METHOD Init_RattlingKM
VAR_INPUT
END_VAR
VAR

END_VAR
                          in_0303_05_1_ixSection1_OverheatAlarm(
	ixSignal:= _0303_05_1_ixSection1_OverheatAlarm, 
	itInputTime:= tRattlingDelay, 
	itRattling_count_reset:= , 
	ixResetAlarm:= , 
	qxSignal=> , 
	qxRattlingAlarm=> );
in_0303_05_1_ixSection1_OverheatWarning(
	ixSignal:= _0303_05_1_ixSection1_OverheatWarning, 
	itInputTime:= tRattlingDelay, 
	itRattling_count_reset:= , 
	ixResetAlarm:= , 
	qxSignal=> , 
	qxRattlingAlarm=> );
in_0303_05_1_ixVFD_Failure(
	ixSignal:= _0303_05_1_ixVFD_Failure, 
	itInputTime:= tRattlingDelay, 
	itRattling_count_reset:= , 
	ixResetAlarm:= , 
	qxSignal=> , 
	qxRattlingAlarm=> );
in_0303_05_1_ixVFD_InWork(
	ixSignal:= _0303_05_1_ixVFD_InWork, 
	itInputTime:= tRattlingDelay, 
	itRattling_count_reset:= , 
	ixResetAlarm:= , 
	qxSignal=> , 
	qxRattlingAlarm=> );
in_0303_05_1_ixVFD_Manual(
	ixSignal:= _0303_05_1_ixVFD_Manual, 
	itInputTime:= tRattlingDelay, 
	itRattling_count_reset:= , 
	ixResetAlarm:= , 
	qxSignal=> , 
	qxRattlingAlarm=> );
in_0303_05_1_ixVFD_Ready(
	ixSignal:= _0303_05_1_ixVFD_Ready, 
	itInputTime:= tRattlingDelay, 
	itRattling_count_reset:= , 
	ixResetAlarm:= , 
	qxSignal=> , 
	qxRattlingAlarm=> );
in_0303_05_2_ixSection1_OverheatAlarm(
	ixSignal:= _0303_05_2_ixSection1_OverheatAlarm, 
	itInputTime:= tRattlingDelay, 
	itRattling_count_reset:= , 
	ixResetAlarm:= , 
	qxSignal=> , 
	qxRattlingAlarm=> );
in_0303_05_2_ixSection1_OverheatWarning(
	ixSignal:= _0303_05_2_ixSection1_OverheatWarning, 
	itInputTime:= tRattlingDelay, 
	itRattling_count_reset:= , 
	ixResetAlarm:= , 
	qxSignal=> , 
	qxRattlingAlarm=> );
in_0303_05_2_ixVFD_Failure(
	ixSignal:= _0303_05_2_ixVFD_Failure, 
	itInputTime:= tRattlingDelay, 
	itRattling_count_reset:= , 
	ixResetAlarm:= , 
	qxSignal=> , 
	qxRattlingAlarm=> );
in_0303_05_2_ixVFD_InWork(
	ixSignal:= _0303_05_2_ixVFD_InWork, 
	itInputTime:= tRattlingDelay, 
	itRattling_count_reset:= , 
	ixResetAlarm:= , 
	qxSignal=> , 
	qxRattlingAlarm=> );
in_0303_05_2_ixVFD_Manual(
	ixSignal:= _0303_05_2_ixVFD_Manual, 
	itInputTime:= tRattlingDelay, 
	itRattling_count_reset:= , 
	ixResetAlarm:= , 
	qxSignal=> , 
	qxRattlingAlarm=> );
in_0303_05_2_ixVFD_Ready(
	ixSignal:= _0303_05_2_ixVFD_Ready, 
	itInputTime:= tRattlingDelay, 
	itRattling_count_reset:= , 
	ixResetAlarm:= , 
	qxSignal=> , 
	qxRattlingAlarm=> );
in_0303_05_1KM8_ixStatusOn(
	ixSignal:= _0303_05_1KM8_ixStatusOn, 
	itInputTime:= tRattlingDelay, 
	itRattling_count_reset:= , 
	ixResetAlarm:= , 
	qxSignal=> , 
	qxRattlingAlarm=> );
in_0303_05_2KM8_ixStatusOn(
	ixSignal:= _0303_05_2KM8_ixStatusOn, 
	itInputTime:= tRattlingDelay, 
	itRattling_count_reset:= , 
	ixResetAlarm:= , 
	qxSignal=> , 
	qxRattlingAlarm=> );
in_0303_05_BY01_ixKM_PosClosed(
	ixSignal:= _0303_05_BY01_ixKM_PosClosed, 
	itInputTime:= tRattlingDelay, 
	itRattling_count_reset:= , 
	ixResetAlarm:= , 
	qxSignal=> , 
	qxRattlingAlarm=> );
in_0303_05_BY01_ixKM_PosOpen(
	ixSignal:= _0303_05_BY01_ixKM_PosOpen, 
	itInputTime:= tRattlingDelay, 
	itRattling_count_reset:= , 
	ixResetAlarm:= , 
	qxSignal=> , 
	qxRattlingAlarm=> );
in_0303_05_BY01_ixShutter_PosClosed(
	ixSignal:= _0303_05_BY01_ixShutter_PosClosed, 
	itInputTime:= tRattlingDelay, 
	itRattling_count_reset:= , 
	ixResetAlarm:= , 
	qxSignal=> , 
	qxRattlingAlarm=> );
in_0303_05_BY01_ixShutter_PosOpen(
	ixSignal:= _0303_05_BY01_ixShutter_PosOpen, 
	itInputTime:= tRattlingDelay, 
	itRattling_count_reset:= , 
	ixResetAlarm:= , 
	qxSignal=> , 
	qxRattlingAlarm=> );
in_0303_05_BY01_ixShutter_StatusError(
	ixSignal:= _0303_05_BY01_ixShutter_StatusError, 
	itInputTime:= tRattlingDelay, 
	itRattling_count_reset:= , 
	ixResetAlarm:= , 
	qxSignal=> , 
	qxRattlingAlarm=> );
in_0303_05_BY01_ixShutter_StatusReady(
	ixSignal:= _0303_05_BY01_ixShutter_StatusReady, 
	itInputTime:= tRattlingDelay, 
	itRattling_count_reset:= , 
	ixResetAlarm:= , 
	qxSignal=> , 
	qxRattlingAlarm=> );
in_0303_05_BY02_ixKM_PosClosed(
	ixSignal:= _0303_05_BY02_ixKM_PosClosed, 
	itInputTime:= tRattlingDelay, 
	itRattling_count_reset:= , 
	ixResetAlarm:= , 
	qxSignal=> , 
	qxRattlingAlarm=> );
in_0303_05_BY02_ixKM_PosOpen(
	ixSignal:= _0303_05_BY02_ixKM_PosOpen, 
	itInputTime:= tRattlingDelay, 
	itRattling_count_reset:= , 
	ixResetAlarm:= , 
	qxSignal=> , 
	qxRattlingAlarm=> );
in_0303_05_BY02_ixShutter_PosClosed(
	ixSignal:= _0303_05_BY02_ixShutter_PosClosed, 
	itInputTime:= tRattlingDelay, 
	itRattling_count_reset:= , 
	ixResetAlarm:= , 
	qxSignal=> , 
	qxRattlingAlarm=> );
in_0303_05_BY02_ixShutter_PosOpen(
	ixSignal:= _0303_05_BY02_ixShutter_PosOpen, 
	itInputTime:= tRattlingDelay, 
	itRattling_count_reset:= , 
	ixResetAlarm:= , 
	qxSignal=> , 
	qxRattlingAlarm=> );
in_0303_05_BY02_ixShutter_StatusError(
	ixSignal:= _0303_05_BY02_ixShutter_StatusError, 
	itInputTime:= tRattlingDelay, 
	itRattling_count_reset:= , 
	ixResetAlarm:= , 
	qxSignal=> , 
	qxRattlingAlarm=> );
in_0303_05_BY02_ixShutter_StatusReady(
	ixSignal:= _0303_05_BY02_ixShutter_StatusReady, 
	itInputTime:= tRattlingDelay, 
	itRattling_count_reset:= , 
	ixResetAlarm:= , 
	qxSignal=> , 
	qxRattlingAlarm=> );
in_0303_05_BY03_ixKM_PosClosed(
	ixSignal:= _0303_05_BY03_ixKM_PosClosed, 
	itInputTime:= tRattlingDelay, 
	itRattling_count_reset:= , 
	ixResetAlarm:= , 
	qxSignal=> , 
	qxRattlingAlarm=> );
in_0303_05_BY03_ixKM_PosOpen(
	ixSignal:= _0303_05_BY03_ixKM_PosOpen, 
	itInputTime:= tRattlingDelay, 
	itRattling_count_reset:= , 
	ixResetAlarm:= , 
	qxSignal=> , 
	qxRattlingAlarm=> );
in_0303_05_BY03_ixShutter_PosClosed(
	ixSignal:= _0303_05_BY03_ixShutter_PosClosed, 
	itInputTime:= tRattlingDelay, 
	itRattling_count_reset:= , 
	ixResetAlarm:= , 
	qxSignal=> , 
	qxRattlingAlarm=> );
in_0303_05_BY03_ixShutter_PosOpen(
	ixSignal:= _0303_05_BY03_ixShutter_PosOpen, 
	itInputTime:= tRattlingDelay, 
	itRattling_count_reset:= , 
	ixResetAlarm:= , 
	qxSignal=> , 
	qxRattlingAlarm=> );
in_0303_05_BY03_ixShutter_StatusError(
	ixSignal:= _0303_05_BY03_ixShutter_StatusError, 
	itInputTime:= tRattlingDelay, 
	itRattling_count_reset:= , 
	ixResetAlarm:= , 
	qxSignal=> , 
	qxRattlingAlarm=> );
in_0303_05_BY03_ixShutter_StatusReady(
	ixSignal:= _0303_05_BY03_ixShutter_StatusReady, 
	itInputTime:= tRattlingDelay, 
	itRattling_count_reset:= , 
	ixResetAlarm:= , 
	qxSignal=> , 
	qxRattlingAlarm=> );
in_0303_05_BY04_ixKM_PosClosed(
	ixSignal:= _0303_05_BY04_ixKM_PosClosed, 
	itInputTime:= tRattlingDelay, 
	itRattling_count_reset:= , 
	ixResetAlarm:= , 
	qxSignal=> , 
	qxRattlingAlarm=> );
in_0303_05_BY04_ixKM_PosOpen(
	ixSignal:= _0303_05_BY04_ixKM_PosOpen, 
	itInputTime:= tRattlingDelay, 
	itRattling_count_reset:= , 
	ixResetAlarm:= , 
	qxSignal=> , 
	qxRattlingAlarm=> );
in_0303_05_BY04_ixShutter_PosClosed(
	ixSignal:= _0303_05_BY04_ixShutter_PosClosed, 
	itInputTime:= tRattlingDelay, 
	itRattling_count_reset:= , 
	ixResetAlarm:= , 
	qxSignal=> , 
	qxRattlingAlarm=> );
in_0303_05_BY04_ixShutter_PosOpen(
	ixSignal:= _0303_05_BY04_ixShutter_PosOpen, 
	itInputTime:= tRattlingDelay, 
	itRattling_count_reset:= , 
	ixResetAlarm:= , 
	qxSignal=> , 
	qxRattlingAlarm=> );
in_0303_05_BY04_ixShutter_StatusError(
	ixSignal:= _0303_05_BY04_ixShutter_StatusError, 
	itInputTime:= tRattlingDelay, 
	itRattling_count_reset:= , 
	ixResetAlarm:= , 
	qxSignal=> , 
	qxRattlingAlarm=> );
in_0303_05_BY04_ixShutter_StatusReady(
	ixSignal:= _0303_05_BY04_ixShutter_StatusReady, 
	itInputTime:= tRattlingDelay, 
	itRattling_count_reset:= , 
	ixResetAlarm:= , 
	qxSignal=> , 
	qxRattlingAlarm=> );
in_0303_05_BY05_ixKM_PosClosed(
	ixSignal:= _0303_05_BY05_ixKM_PosClosed, 
	itInputTime:= tRattlingDelay, 
	itRattling_count_reset:= , 
	ixResetAlarm:= , 
	qxSignal=> , 
	qxRattlingAlarm=> );
in_0303_05_BY05_ixKM_PosOpen(
	ixSignal:= _0303_05_BY05_ixKM_PosOpen, 
	itInputTime:= tRattlingDelay, 
	itRattling_count_reset:= , 
	ixResetAlarm:= , 
	qxSignal=> , 
	qxRattlingAlarm=> );
in_0303_05_BY05_ixShutter_PosClosed(
	ixSignal:= _0303_05_BY05_ixShutter_PosClosed, 
	itInputTime:= tRattlingDelay, 
	itRattling_count_reset:= , 
	ixResetAlarm:= , 
	qxSignal=> , 
	qxRattlingAlarm=> );
in_0303_05_BY05_ixShutter_PosOpen(
	ixSignal:= _0303_05_BY05_ixShutter_PosOpen, 
	itInputTime:= tRattlingDelay, 
	itRattling_count_reset:= , 
	ixResetAlarm:= , 
	qxSignal=> , 
	qxRattlingAlarm=> );
in_0303_05_BY05_ixShutter_StatusError(
	ixSignal:= _0303_05_BY05_ixShutter_StatusError, 
	itInputTime:= tRattlingDelay, 
	itRattling_count_reset:= , 
	ixResetAlarm:= , 
	qxSignal=> , 
	qxRattlingAlarm=> );
in_0303_05_BY05_ixShutter_StatusReady(
	ixSignal:= _0303_05_BY05_ixShutter_StatusReady, 
	itInputTime:= tRattlingDelay, 
	itRattling_count_reset:= , 
	ixResetAlarm:= , 
	qxSignal=> , 
	qxRattlingAlarm=> );
in_0303_05_BY07_ixKM_PosClosed(
	ixSignal:= _0303_05_BY07_ixKM_PosClosed, 
	itInputTime:= tRattlingDelay, 
	itRattling_count_reset:= , 
	ixResetAlarm:= , 
	qxSignal=> , 
	qxRattlingAlarm=> );
in_0303_05_BY07_ixKM_PosOpen(
	ixSignal:= _0303_05_BY07_ixKM_PosOpen, 
	itInputTime:= tRattlingDelay, 
	itRattling_count_reset:= , 
	ixResetAlarm:= , 
	qxSignal=> , 
	qxRattlingAlarm=> );
in_0303_05_BY07_ixShutter_PosClosed(
	ixSignal:= _0303_05_BY07_ixShutter_PosClosed, 
	itInputTime:= tRattlingDelay, 
	itRattling_count_reset:= , 
	ixResetAlarm:= , 
	qxSignal=> , 
	qxRattlingAlarm=> );
in_0303_05_BY07_ixShutter_PosOpen(
	ixSignal:= _0303_05_BY07_ixShutter_PosOpen, 
	itInputTime:= tRattlingDelay, 
	itRattling_count_reset:= , 
	ixResetAlarm:= , 
	qxSignal=> , 
	qxRattlingAlarm=> );
in_0303_05_BY07_ixShutter_StatusError(
	ixSignal:= _0303_05_BY07_ixShutter_StatusError, 
	itInputTime:= tRattlingDelay, 
	itRattling_count_reset:= , 
	ixResetAlarm:= , 
	qxSignal=> , 
	qxRattlingAlarm=> );
in_0303_05_BY07_ixShutter_StatusReady(
	ixSignal:= _0303_05_BY07_ixShutter_StatusReady, 
	itInputTime:= tRattlingDelay, 
	itRattling_count_reset:= , 
	ixResetAlarm:= , 
	qxSignal=> , 
	qxRattlingAlarm=> );
in_0303_05_BY08_ixKM_PosClosed(
	ixSignal:= _0303_05_BY08_ixKM_PosClosed, 
	itInputTime:= tRattlingDelay, 
	itRattling_count_reset:= , 
	ixResetAlarm:= , 
	qxSignal=> , 
	qxRattlingAlarm=> );
in_0303_05_BY08_ixKM_PosOpen(
	ixSignal:= _0303_05_BY08_ixKM_PosOpen, 
	itInputTime:= tRattlingDelay, 
	itRattling_count_reset:= , 
	ixResetAlarm:= , 
	qxSignal=> , 
	qxRattlingAlarm=> );
in_0303_05_BY08_ixShutter_PosClosed(
	ixSignal:= _0303_05_BY08_ixShutter_PosClosed, 
	itInputTime:= tRattlingDelay, 
	itRattling_count_reset:= , 
	ixResetAlarm:= , 
	qxSignal=> , 
	qxRattlingAlarm=> );
in_0303_05_BY08_ixShutter_PosOpen(
	ixSignal:= _0303_05_BY08_ixShutter_PosOpen, 
	itInputTime:= tRattlingDelay, 
	itRattling_count_reset:= , 
	ixResetAlarm:= , 
	qxSignal=> , 
	qxRattlingAlarm=> );
in_0303_05_BY08_ixShutter_StatusError(
	ixSignal:= _0303_05_BY08_ixShutter_StatusError, 
	itInputTime:= tRattlingDelay, 
	itRattling_count_reset:= , 
	ixResetAlarm:= , 
	qxSignal=> , 
	qxRattlingAlarm=> );
in_0303_05_BY08_ixShutter_StatusReady(
	ixSignal:= _0303_05_BY08_ixShutter_StatusReady, 
	itInputTime:= tRattlingDelay, 
	itRattling_count_reset:= , 
	ixResetAlarm:= , 
	qxSignal=> , 
	qxRattlingAlarm=> );
in_0303_05_PU01_ixKM_StatusManualStart(
	ixSignal:= _0303_05_PU01_ixKM_StatusManualStart, 
	itInputTime:= tRattlingDelay, 
	itRattling_count_reset:= , 
	ixResetAlarm:= , 
	qxSignal=> , 
	qxRattlingAlarm=> );
in_0303_05_PU01_ixKM_StatusManualStop(
	ixSignal:= _0303_05_PU01_ixKM_StatusManualStop, 
	itInputTime:= tRattlingDelay, 
	itRattling_count_reset:= , 
	ixResetAlarm:= , 
	qxSignal=> , 
	qxRattlingAlarm=> );
in_0303_05_PU01_ixKM_StatusOn(
	ixSignal:= _0303_05_PU01_ixKM_StatusOn, 
	itInputTime:= tRattlingDelay, 
	itRattling_count_reset:= , 
	ixResetAlarm:= , 
	qxSignal=> , 
	qxRattlingAlarm=> );
in_0303_05_PU01_ixKM_VFD_StatusOn(
	ixSignal:= _0303_05_PU01_ixKM_VFD_StatusOn, 
	itInputTime:= tRattlingDelay, 
	itRattling_count_reset:= , 
	ixResetAlarm:= , 
	qxSignal=> , 
	qxRattlingAlarm=> );
in_0303_05_PU01_ixStatusManual(
	ixSignal:= _0303_05_PU01_ixStatusManual, 
	itInputTime:= tRattlingDelay, 
	itRattling_count_reset:= , 
	ixResetAlarm:= , 
	qxSignal=> , 
	qxRattlingAlarm=> );
in_0303_05_PU02_ixKM_StatusManualStart(
	ixSignal:= _0303_05_PU02_ixKM_StatusManualStart, 
	itInputTime:= tRattlingDelay, 
	itRattling_count_reset:= , 
	ixResetAlarm:= , 
	qxSignal=> , 
	qxRattlingAlarm=> );
in_0303_05_PU02_ixKM_StatusManualStop(
	ixSignal:= _0303_05_PU02_ixKM_StatusManualStop, 
	itInputTime:= tRattlingDelay, 
	itRattling_count_reset:= , 
	ixResetAlarm:= , 
	qxSignal=> , 
	qxRattlingAlarm=> );
in_0303_05_PU02_ixKM_StatusOn(
	ixSignal:= _0303_05_PU02_ixKM_StatusOn, 
	itInputTime:= tRattlingDelay, 
	itRattling_count_reset:= , 
	ixResetAlarm:= , 
	qxSignal=> , 
	qxRattlingAlarm=> );
in_0303_05_PU02_ixKM_VFD_StatusOn(
	ixSignal:= _0303_05_PU02_ixKM_VFD_StatusOn, 
	itInputTime:= tRattlingDelay, 
	itRattling_count_reset:= , 
	ixResetAlarm:= , 
	qxSignal=> , 
	qxRattlingAlarm=> );
in_0303_05_PU02_ixStatusManual(
	ixSignal:= _0303_05_PU02_ixStatusManual, 
	itInputTime:= tRattlingDelay, 
	itRattling_count_reset:= , 
	ixResetAlarm:= , 
	qxSignal=> , 
	qxRattlingAlarm=> );
in_0303_05_PU03_ixKM_StatusManualStart(
	ixSignal:= _0303_05_PU03_ixKM_StatusManualStart, 
	itInputTime:= tRattlingDelay, 
	itRattling_count_reset:= , 
	ixResetAlarm:= , 
	qxSignal=> , 
	qxRattlingAlarm=> );
in_0303_05_PU03_ixKM_StatusManualStop(
	ixSignal:= _0303_05_PU03_ixKM_StatusManualStop, 
	itInputTime:= tRattlingDelay, 
	itRattling_count_reset:= , 
	ixResetAlarm:= , 
	qxSignal=> , 
	qxRattlingAlarm=> );
in_0303_05_PU03_ixKM_StatusOn(
	ixSignal:= _0303_05_PU03_ixKM_StatusOn, 
	itInputTime:= tRattlingDelay, 
	itRattling_count_reset:= , 
	ixResetAlarm:= , 
	qxSignal=> , 
	qxRattlingAlarm=> );
in_0303_05_PU03_ixKM_VFD_StatusOn(
	ixSignal:= _0303_05_PU03_ixKM_VFD_StatusOn, 
	itInputTime:= tRattlingDelay, 
	itRattling_count_reset:= , 
	ixResetAlarm:= , 
	qxSignal=> , 
	qxRattlingAlarm=> );
in_0303_05_PU03_ixStatusManual(
	ixSignal:= _0303_05_PU03_ixStatusManual, 
	itInputTime:= tRattlingDelay, 
	itRattling_count_reset:= , 
	ixResetAlarm:= , 
	qxSignal=> , 
	qxRattlingAlarm=> );
in_0303_05_PU04_ixKM_StatusManualStart(
	ixSignal:= _0303_05_PU04_ixKM_StatusManualStart, 
	itInputTime:= tRattlingDelay, 
	itRattling_count_reset:= , 
	ixResetAlarm:= , 
	qxSignal=> , 
	qxRattlingAlarm=> );
in_0303_05_PU04_ixKM_StatusManualStop(
	ixSignal:= _0303_05_PU04_ixKM_StatusManualStop, 
	itInputTime:= tRattlingDelay, 
	itRattling_count_reset:= , 
	ixResetAlarm:= , 
	qxSignal=> , 
	qxRattlingAlarm=> );
in_0303_05_PU04_ixKM_StatusOn(
	ixSignal:= _0303_05_PU04_ixKM_StatusOn, 
	itInputTime:= tRattlingDelay, 
	itRattling_count_reset:= , 
	ixResetAlarm:= , 
	qxSignal=> , 
	qxRattlingAlarm=> );
in_0303_05_PU04_ixKM_VFD_StatusOn(
	ixSignal:= _0303_05_PU04_ixKM_VFD_StatusOn, 
	itInputTime:= tRattlingDelay, 
	itRattling_count_reset:= , 
	ixResetAlarm:= , 
	qxSignal=> , 
	qxRattlingAlarm=> );
in_0303_05_PU04_ixStatusManual(
	ixSignal:= _0303_05_PU04_ixStatusManual, 
	itInputTime:= tRattlingDelay, 
	itRattling_count_reset:= , 
	ixResetAlarm:= , 
	qxSignal=> , 
	qxRattlingAlarm=> );
in_0303_05_PU05_ixKM_StatusManualStart(
	ixSignal:= _0303_05_PU05_ixKM_StatusManualStart, 
	itInputTime:= tRattlingDelay, 
	itRattling_count_reset:= , 
	ixResetAlarm:= , 
	qxSignal=> , 
	qxRattlingAlarm=> );
in_0303_05_PU05_ixKM_StatusManualStop(
	ixSignal:= _0303_05_PU05_ixKM_StatusManualStop, 
	itInputTime:= tRattlingDelay, 
	itRattling_count_reset:= , 
	ixResetAlarm:= , 
	qxSignal=> , 
	qxRattlingAlarm=> );
in_0303_05_PU05_ixKM_StatusOn(
	ixSignal:= _0303_05_PU05_ixKM_StatusOn, 
	itInputTime:= tRattlingDelay, 
	itRattling_count_reset:= , 
	ixResetAlarm:= , 
	qxSignal=> , 
	qxRattlingAlarm=> );
in_0303_05_PU05_ixKM_VFD_StatusOn(
	ixSignal:= _0303_05_PU05_ixKM_VFD_StatusOn, 
	itInputTime:= tRattlingDelay, 
	itRattling_count_reset:= , 
	ixResetAlarm:= , 
	qxSignal=> , 
	qxRattlingAlarm=> );
in_0303_05_PU05_ixStatusManual(
	ixSignal:= _0303_05_PU05_ixStatusManual, 
	itInputTime:= tRattlingDelay, 
	itRattling_count_reset:= , 
	ixResetAlarm:= , 
	qxSignal=> , 
	qxRattlingAlarm=> );

                        
END_METHOD

METHOD Initialization
VAR_INPUT
END_VAR
                          Init_VFD_Main();
Init_VFD_Reserve();

Init_RattlingKM();
Init_ServiceAutoSignals();
Init_triggers();
                        
END_METHOD

METHOD GetStatus_PU_VFD : BOOL
VAR_INPUT
	i : INT;
END_VAR
                          CASE i OF
	1:	GetStatus_PU_VFD := in_0303_05_PU01_ixKM_VFD_StatusOn.qxSignal;
	2:	GetStatus_PU_VFD := in_0303_05_PU02_ixKM_VFD_StatusOn.qxSignal;
	3:	GetStatus_PU_VFD := in_0303_05_PU03_ixKM_VFD_StatusOn.qxSignal;
	4:	GetStatus_PU_VFD := in_0303_05_PU04_ixKM_VFD_StatusOn.qxSignal;
	5:	GetStatus_PU_VFD := in_0303_05_PU05_ixKM_VFD_StatusOn.qxSignal;
END_CASE;
                        
END_METHOD

METHOD GetStatus_PU_BP : BOOL
VAR_INPUT
	i : INT;
END_VAR
                          CASE i OF
	1:	GetStatus_PU_BP := in_0303_05_PU01_ixKM_StatusOn.qxSignal;
	2:	GetStatus_PU_BP := in_0303_05_PU02_ixKM_StatusOn.qxSignal;
	3:	GetStatus_PU_BP := in_0303_05_PU03_ixKM_StatusOn.qxSignal;
	4:	GetStatus_PU_BP := in_0303_05_PU04_ixKM_StatusOn.qxSignal;
	5:	GetStatus_PU_BP := in_0303_05_PU05_ixKM_StatusOn.qxSignal;
END_CASE;
                        
END_METHOD

METHOD GetStatus_BY_Open : BOOL
VAR_INPUT
	i : INT;
END_VAR
                          CASE i OF
	1:	GetStatus_BY_Open := in_0303_05_BY01_ixShutter_PosOpen.qxSignal;
	2:	GetStatus_BY_Open := in_0303_05_BY02_ixShutter_PosOpen.qxSignal;
	3:	GetStatus_BY_Open := in_0303_05_BY03_ixShutter_PosOpen.qxSignal;
	4:	GetStatus_BY_Open := in_0303_05_BY04_ixShutter_PosOpen.qxSignal;
	5:	GetStatus_BY_Open := in_0303_05_BY05_ixShutter_PosOpen.qxSignal;
	7:	GetStatus_BY_Open := in_0303_05_BY07_ixShutter_PosOpen.qxSignal;
	8:	GetStatus_BY_Open := in_0303_05_BY08_ixShutter_PosOpen.qxSignal;
END_CASE;
                        
END_METHOD

METHOD GetStatus_BY_Closed : BOOL
VAR_INPUT
	i : INT;
END_VAR
                          CASE i OF
	1:	GetStatus_BY_Closed := in_0303_05_BY01_ixShutter_PosClosed.qxSignal;
	2:	GetStatus_BY_Closed := in_0303_05_BY02_ixShutter_PosClosed.qxSignal;
	3:	GetStatus_BY_Closed := in_0303_05_BY03_ixShutter_PosClosed.qxSignal;
	4:	GetStatus_BY_Closed := in_0303_05_BY04_ixShutter_PosClosed.qxSignal;
	5:	GetStatus_BY_Closed := in_0303_05_BY05_ixShutter_PosClosed.qxSignal;
	7:	GetStatus_BY_Closed := in_0303_05_BY07_ixShutter_PosClosed.qxSignal;
	8:	GetStatus_BY_Closed := in_0303_05_BY08_ixShutter_PosClosed.qxSignal;
END_CASE;
                        
END_METHOD

METHOD GetStatus_BY_Ready : BOOL
VAR_INPUT
	i : INT;
END_VAR
                          CASE i OF
	1:	GetStatus_BY_Ready := in_0303_05_BY01_ixShutter_StatusReady.qxSignal;
	2:	GetStatus_BY_Ready := in_0303_05_BY02_ixShutter_StatusReady.qxSignal;
	3:	GetStatus_BY_Ready := in_0303_05_BY03_ixShutter_StatusReady.qxSignal;
	4:	GetStatus_BY_Ready := in_0303_05_BY04_ixShutter_StatusReady.qxSignal;
	5:	GetStatus_BY_Ready := in_0303_05_BY05_ixShutter_StatusReady.qxSignal;
	7:	GetStatus_BY_Ready := in_0303_05_BY07_ixShutter_StatusReady.qxSignal;
	8:	GetStatus_BY_Ready := in_0303_05_BY08_ixShutter_StatusReady.qxSignal;
END_CASE;
                        
END_METHOD

METHOD GetStatus_BY_Error : BOOL
VAR_INPUT
	i : INT;
END_VAR
                          CASE i OF
	1:	GetStatus_BY_Error := in_0303_05_BY01_ixShutter_StatusError.qxSignal;
	2:	GetStatus_BY_Error := in_0303_05_BY02_ixShutter_StatusError.qxSignal;
	3:	GetStatus_BY_Error := in_0303_05_BY03_ixShutter_StatusError.qxSignal;
	4:	GetStatus_BY_Error := in_0303_05_BY04_ixShutter_StatusError.qxSignal;
	5:	GetStatus_BY_Error := in_0303_05_BY05_ixShutter_StatusError.qxSignal;
	7:	GetStatus_BY_Error := in_0303_05_BY07_ixShutter_StatusError.qxSignal;
	8:	GetStatus_BY_Error := in_0303_05_BY08_ixShutter_StatusError.qxSignal;
END_CASE;
                        
END_METHOD

METHOD Set_BY_Open
VAR_INPUT
	i : INT;
	x : BOOL;
END_VAR
                          CASE i OF
	1: _0303_05_BY01_qxShutter_Open := x;
	2: _0303_05_BY02_qxShutter_Open := x;
	3: _0303_05_BY03_qxShutter_Open := x;
	4: _0303_05_BY04_qxShutter_Open := x;
	5: _0303_05_BY05_qxShutter_Open := x;
	7: _0303_05_BY07_qxShutter_Open := x;
	8: _0303_05_BY08_qxShutter_Open := x;
END_CASE;
                        
END_METHOD

METHOD Set_BY_Close
VAR_INPUT
	i : INT;
	x : BOOL;
END_VAR
                          CASE i OF
	1: _0303_05_BY01_qxShutter_Close := x;
	2: _0303_05_BY02_qxShutter_Close := x;
	3: _0303_05_BY03_qxShutter_Close := x;
	4: _0303_05_BY04_qxShutter_Close := x;
	5: _0303_05_BY05_qxShutter_Close := x;
	7: _0303_05_BY07_qxShutter_Close := x;
	8: _0303_05_BY08_qxShutter_Close := x;
END_CASE;
                        
END_METHOD

METHOD Set_PU_VFD
VAR_INPUT
	i : INT;
	x : BOOL;
END_VAR
                          CASE i OF
	1: _0303_05_PU01_qxKM_Frq_cmdOn := x;
	2: _0303_05_PU02_qxKM_Frq_cmdOn := x;
	3: _0303_05_PU03_qxKM_Frq_cmdOn := x;
	4: _0303_05_PU04_qxKM_Frq_cmdOn := x;
	5: _0303_05_PU05_qxKM_Frq_cmdOn := x;
END_CASE;
                        
END_METHOD

METHOD Set_PU_BP
VAR_INPUT
	i : INT;
	x : BOOL;
END_VAR
                          CASE i OF
	1: _0303_05_PU01_qxKM_cmdOn := x;
	2: _0303_05_PU02_qxKM_cmdOn := x;
	3: _0303_05_PU03_qxKM_cmdOn := x;
	4: _0303_05_PU04_qxKM_cmdOn := x;
	5: _0303_05_PU05_qxKM_cmdOn := x;
END_CASE;
                        
END_METHOD

METHOD Set_KM8
VAR_INPUT
	i : INT;
	x : BOOL;
END_VAR
                          CASE i OF
	1: IF NOT _0303_05_2KM8_qxOn THEN _0303_05_1KM8_qxOn := x; END_IF;
	2: IF NOT _0303_05_1KM8_qxOn THEN _0303_05_2KM8_qxOn := x; END_IF;
END_CASE;
                        
END_METHOD

METHOD Set_PU_DryRun
VAR_INPUT
	i : INT;
	x : BOOL;
END_VAR
                          CASE i OF
	1: _0303_05_PU01_qxDryRun := x;
	2: _0303_05_PU02_qxDryRun := x;
	3: _0303_05_PU03_qxDryRun := x;
	4: _0303_05_PU04_qxDryRun := x;
	5: _0303_05_PU05_qxDryRun := x;
END_CASE;
                        
END_METHOD

METHOD GetStatus_PU_Manual : BOOL
VAR_INPUT
	i : INT;
END_VAR
                          CASE i OF
	1:	GetStatus_PU_Manual := in_0303_05_PU01_ixStatusManual.qxSignal;
	2:	GetStatus_PU_Manual := in_0303_05_PU02_ixStatusManual.qxSignal;
	3:	GetStatus_PU_Manual := in_0303_05_PU03_ixStatusManual.qxSignal;
	4:	GetStatus_PU_Manual := in_0303_05_PU04_ixStatusManual.qxSignal;
	5:	GetStatus_PU_Manual := in_0303_05_PU05_ixStatusManual.qxSignal;
END_CASE;
                        
END_METHOD

METHOD GetStatus_PU_VFD_ManualStart : BOOL
VAR_INPUT
	i : INT;
END_VAR
                          CASE i OF
	1:	GetStatus_PU_VFD_ManualStart := in_0303_05_PU01_ixKM_StatusManualStart.qxSignal;
	2:	GetStatus_PU_VFD_ManualStart := in_0303_05_PU02_ixKM_StatusManualStart.qxSignal;
	3:	GetStatus_PU_VFD_ManualStart := in_0303_05_PU03_ixKM_StatusManualStart.qxSignal;
	4:	GetStatus_PU_VFD_ManualStart := in_0303_05_PU04_ixKM_StatusManualStart.qxSignal;
	5:	GetStatus_PU_VFD_ManualStart := in_0303_05_PU05_ixKM_StatusManualStart.qxSignal;
END_CASE;
                        
END_METHOD

METHOD GetStatus_PU_VFD_ManualStop : BOOL
VAR_INPUT
	i : INT;
END_VAR
                          CASE i OF
	1:	GetStatus_PU_VFD_ManualStop := in_0303_05_PU01_ixKM_StatusManualStop.qxSignal;
	2:	GetStatus_PU_VFD_ManualStop := in_0303_05_PU02_ixKM_StatusManualStop.qxSignal;
	3:	GetStatus_PU_VFD_ManualStop := in_0303_05_PU03_ixKM_StatusManualStop.qxSignal;
	4:	GetStatus_PU_VFD_ManualStop := in_0303_05_PU04_ixKM_StatusManualStop.qxSignal;
	5:	GetStatus_PU_VFD_ManualStop := in_0303_05_PU05_ixKM_StatusManualStop.qxSignal;
END_CASE;
                        
END_METHOD

METHOD GetStatus_VFD_Error : BOOL
VAR_INPUT
	i : INT;
END_VAR
                          CASE i OF
	1: GetStatus_VFD_Error := in_0303_05_1_ixVFD_Failure.qxSignal;
	2: GetStatus_VFD_Error := in_0303_05_2_ixVFD_Failure.qxSignal;
END_CASE;
                        
END_METHOD

METHOD GetStatus_VFD_Ready : BOOL
VAR_INPUT
	i : INT;
END_VAR
                          CASE i OF
	1: GetStatus_VFD_Ready := in_0303_05_1_ixVFD_Ready.qxSignal;
	2: GetStatus_VFD_Ready := in_0303_05_2_ixVFD_Ready.qxSignal;
END_CASE;
                        
END_METHOD

METHOD GetStatus_VFD_ActualFreq : REAL
VAR_INPUT
	i : INT;
END_VAR
                          CASE i OF
	1: GetStatus_VFD_ActualFreq := _0303_05_VFD001_MainVFD_ActualFrequency.Value;
	2: GetStatus_VFD_ActualFreq := _0303_05_VFD002_ReserveVFD_ActualFrequency.Value;
END_CASE;
                        
END_METHOD

METHOD Set_VFD_Change
VAR_INPUT
	i : INT;
END_VAR
                          vfd_iChange := i;
                        
END_METHOD

METHOD Process_VFD_qFreq
VAR_INPUT
END_VAR
                          // Задание частоты на модуль аналогового выхода, зависимо от выбранного ЧРП
Set_VFD_OutSignalToModule(
	vfd_iChange,
	GetValue_VFD_OutSignalConvertation(GetValue_VFD_qrFreq(vfd_iChange))
);
                        
END_METHOD

METHOD GetValue_VFD_OutSignalConvertation : UINT
VAR_INPUT
	rValue : REAL;
END_VAR
VAR
	A_Signal_Output : FB_Asignal_FreqConvertation;
END_VAR
                          A_Signal_Output(
	irSetFrequencyHz:= rValue, 
	irSetFrequencyHzMax:= vfd_rMaxFreq, 
	qIScaledValue=> GetValue_VFD_OutSignalConvertation);
                        
END_METHOD

METHOD Set_VFD_OutSignalToModule // Задание частоты на выбранный модуль аналогового выхода
VAR_INPUT
	iChange : INT;
	iValue : UINT;
END_VAR
                          CASE iChange OF
	1: _0303_05_VFD001_qIMainFrq_SetFrq := iValue;
	2: _0303_05_VFD002_qIReserveFrq_SetFrq := iValue;
END_CASE;
                        
END_METHOD

METHOD GetValue_VFD_qrFreq : REAL
VAR_INPUT
	i : INT;
END_VAR
                          CASE i OF
	1: GetValue_VFD_qrFreq := VFD_MAIN.qrFreq;
	2: GetValue_VFD_qrFreq := VFD_RESERVE.qrFreq;
END_CASE;
                        
END_METHOD

METHOD Process_VFD_Commands
VAR_INPUT
	xStart : BOOL;
	xStop : BOOL;
	xEmergencyStop : BOOL;
	xReset : BOOL;
END_VAR
VAR
	ftrig_xReset : F_TRIG;
END_VAR
                          // Старт насоса от ЧРП
IF xStart AND Condition_PU_toVFD(vfd_iChange, pu_iChange) THEN
	Set_KM8(vfd_iChange, TRUE);
	Set_VFD_Start(vfd_iChange, TRUE);
	Set_PU_VFD(pu_iChange, TRUE);
END_IF;

// Стоп насосса от ЧРП
IF xStop THEN
	Set_VFD_Stop(pu_iChange, FALSE);
	Set_PU_VFD(pu_iChange, FALSE);
	Set_KM8(vfd_iChange, FALSE);
END_IF;

// Аварийная остановка ЧРП
IF xEmergencyStop THEN
	Set_VFD_EmergencyStop(vfd_iChange, TRUE);
END_IF;

// Работа сброса ошибок ФБ ЧРП
ftrig_xReset(CLK:= xReset, Q=> );
IF xReset THEN
	Set_VFD_Reset(vfd_iChange, TRUE);
END_IF;
IF ftrig_xReset.Q THEN Set_VFD_Reset(vfd_iChange, FALSE); END_IF;


                        
END_METHOD

METHOD Set_VFD_Start
VAR_INPUT
	i : INT;
	x : BOOL;
END_VAR
                          CASE i OF
	1: VFD_MAIN.ixStart := x;
	2: VFD_RESERVE.ixStart := x;
END_CASE;
                        
END_METHOD

METHOD Set_VFD_Stop
VAR_INPUT
	i : INT;
	x : BOOL;
END_VAR
                          CASE i OF
	1: VFD_MAIN.ixStop := x;
	2: VFD_RESERVE.ixStop := x;
END_CASE;
                        
END_METHOD

METHOD Set_VFD_FastStart
VAR_INPUT
	i : INT;
	x : BOOL;
END_VAR
                          CASE i OF
	1: VFD_MAIN.ixFastStart := x;
	2: VFD_RESERVE.ixFastStart := x;
END_CASE;
                        
END_METHOD

METHOD Set_VFD_EmergencyStop
VAR_INPUT
	i : INT;
	x : BOOL;
END_VAR
                          CASE i OF
	1: VFD_MAIN.ixEmergencyStop := x;
	2: VFD_RESERVE.ixEmergencyStop := x;
END_CASE;
                        
END_METHOD

METHOD Set_VFD_Reset
VAR_INPUT
	i : INT;
	x : BOOL;
END_VAR
                          CASE i OF
	1: VFD_MAIN.ixReset := x;
	2: VFD_RESERVE.ixReset := x;
END_CASE;
                        
END_METHOD

METHOD GetStatus_VFD_qStart : BOOL
VAR_INPUT
	i : INT;
END_VAR
                          CASE i OF
	1: GetStatus_VFD_qStart := VFD_MAIN.qxStart;
	2: GetStatus_VFD_qStart := VFD_RESERVE.qxStart;
END_CASE;
                        
END_METHOD

METHOD GetStatus_VFD_qStop : BOOL
VAR_INPUT
	i : INT;
END_VAR
                          CASE i OF
	1: GetStatus_VFD_qStop := VFD_MAIN.qxStop;
	2: GetStatus_VFD_qStop := VFD_RESERVE.qxStop;
END_CASE;
                        
END_METHOD

METHOD GetStatus_VFD_qEmergencyStopStatus : BOOL
VAR_INPUT
	i : INT;
END_VAR
                          CASE i OF
	1: GetStatus_VFD_qEmergencyStopStatus := VFD_MAIN.qxEmergencyStopStatus;
	2: GetStatus_VFD_qEmergencyStopStatus := VFD_RESERVE.qxEmergencyStopStatus;
END_CASE;
                        
END_METHOD

METHOD GetStatus_VFD_qErrorInvalidInaccuracy : BOOL
VAR_INPUT
	i : INT;
END_VAR
                          CASE i OF
	1: GetStatus_VFD_qErrorInvalidInaccuracy := VFD_MAIN.qxErrorInvalidInaccuracy;
	2: GetStatus_VFD_qErrorInvalidInaccuracy := VFD_RESERVE.qxErrorInvalidInaccuracy;
END_CASE;
                        
END_METHOD

METHOD GetStatus_VFD_qDelayError : BOOL
VAR_INPUT
	i : INT;
END_VAR
                          CASE i OF
	1: GetStatus_VFD_qDelayError := VFD_MAIN.qxDelayError;
	2: GetStatus_VFD_qDelayError := VFD_RESERVE.qxDelayError;
END_CASE;
                        
END_METHOD

METHOD Condition_PU_toBP : BOOL
VAR_INPUT
	i : INT;
END_VAR
                          Condition_PU_toBP :=
	NOT GetStatus_PU_BP(i)
	AND NOT GetStatus_PU_VFD(i);
                        
END_METHOD

METHOD Condition_PU_toVFD : BOOL
VAR_INPUT
	VFD : INT;
	PU : INT;
	
END_VAR
                          Condition_PU_toVFD := 
	GetStatus_VFD_Ready(VFD)
	AND NOT GetStatus_PU_VFD_Common()
	AND NOT GetStatus_PU_Manual(PU)
	AND NOT GetStatus_PU_BP(PU);

                        
END_METHOD

METHOD GetStatus_PU_VFD_Common : BOOL
VAR_INPUT
END_VAR
                          GetStatus_PU_VFD_Common := 
	in_0303_05_PU01_ixKM_VFD_StatusOn.qxSignal
	OR in_0303_05_PU02_ixKM_VFD_StatusOn.qxSignal
	OR in_0303_05_PU03_ixKM_VFD_StatusOn.qxSignal
	OR in_0303_05_PU04_ixKM_VFD_StatusOn.qxSignal
	OR in_0303_05_PU05_ixKM_VFD_StatusOn.qxSignal;

                        
END_METHOD

METHOD Set_PU_Change
VAR_INPUT
	i : INT;
END_VAR
                          pu_iChange := i;
                        
END_METHOD

METHOD Process_PU_Commands
VAR_INPUT
	xStart : BOOL;
	xStop : BOOL;
	xReset : BOOL;
	xChange_VFDtoBP : BOOL;
	xChange_BPtoVFD : BOOL;
END_VAR
VAR
END_VAR
                          // IF xReset THEN
// 	
// END_IF;


// Запуск по команде на БП
IF xStart AND Condition_PU_toBP(pu_iChange) THEN
	Set_PU_BP(pu_iChange, TRUE);
END_IF;

IF xStop AND Condition_PU_toBP(pu_iChange) THEN
	Set_PU_BP(pu_iChange, FALSE);
END_IF;

// Работа смены ЧРП и БП
IF xChange_VFDtoBP THEN
	Set_PU_VFD(pu_iChange, FALSE);	
	Set_PU_BP(pu_iChange, TRUE);
END_IF;

IF xChange_BPtoVFD AND NOT GetStatus_PU_VFD_Common() THEN
	Set_PU_BP(pu_iChange, FALSE);
	Set_PU_VFD(pu_iChange, TRUE);	
END_IF;

                        
END_METHOD

METHOD Process_PU_Signals
VAR_INPUT
END_VAR
                          // Set_PU_VFD(pu_iChange, GetStatus_VFD_qStart(vfd_iChange));

                        
END_METHOD

METHOD Set_VFD_ChangeFrq
VAR_INPUT
	frq : REAL;
END_VAR
                          vfd_rSetFreq := frq;
                        
END_METHOD

METHOD Process_PU
VAR_INPUT
END_VAR
                          Process_PU_Commands(
	rtrig_puCmd_xStart.Q,
	rtrig_puCmd_xStop.Q,
	rtrig_puCmd_xReset.Q,
	rtrig_puCmd_xChange_VFDtoBP.Q,
	rtrig_puCmd_xChange_BPtoVFD.Q
);
Process_PU_Signals();
                        
END_METHOD

METHOD Process_VFD_Signals
VAR_INPUT
END_VAR
                          IF NOT GetStatus_PU_VFD_Common() THEN
	Set_KM8(vfd_iChange, FALSE);
END_IF;
                        
END_METHOD

METHOD Init_triggers
VAR_INPUT
END_VAR
VAR
END_VAR
                          rtrig_puCmd_xStart(CLK:= xPU_Start.qxSignal, Q=> );
rtrig_puCmd_xStop(CLK:= xPU_Stop.qxSignal, Q=> );
rtrig_puCmd_xReset(CLK:= xPU_Reset.qxSignal, Q=> );
rtrig_puCmd_xChange_VFDtoBP(CLK:= xPU_Change_VFDtoBP.qxSignal, Q=> );
rtrig_puCmd_xChange_BPtoVFD(CLK:= xPU_Change_BPtoVFD.qxSignal, Q=> );

rtrig_vfdCmd_xStart(CLK:= xVFD_Start.qxSignal, Q=> );
rtrig_vfdCmd_xEmergencyStop(CLK:= xVFD_Start.qxSignal, Q=> );
rtrig_vfdCmd_xStop(CLK:= xVFD_Stop.qxSignal, Q=> );
rtrig_vfdCmd_xReset(CLK:= xVFD_Reset.qxSignal, Q=> );

rtrig_byCmd_xOpen(CLK:= xBY_Open.qxSignal, Q=> );
rtrig_byCmd_xClose(CLK:= xBY_Close.qxSignal, Q=> );
rtrig_byCmd_xStop(CLK:= xBY_Stop.qxSignal, Q=> );
rtrig_byCmd_xReset(CLK:= xBY_Close.qxSignal, Q=> );

                        
END_METHOD

METHOD Init_ServiceAutoSignals
VAR_INPUT
END_VAR
                          // КОМАНДЫ - НАСОС
xPU_Start(
	ixAutoSignal:= , 
	ixServiceSignal:= , 
	iiPLCMode:= PLC_Mode, 
	qxSignal=> );

xPU_Stop(
	ixAutoSignal:= , 
	ixServiceSignal:= , 
	iiPLCMode:= PLC_Mode, 
	qxSignal=> );

xPU_Reset(
	ixAutoSignal:= , 
	ixServiceSignal:= , 
	iiPLCMode:= PLC_Mode, 
	qxSignal=> );

xPU_Change_VFDtoBP(
	ixAutoSignal:= , 
	ixServiceSignal:= , 
	iiPLCMode:= PLC_Mode, 
	qxSignal=> );

xPU_Change_BPtoVFD(
	ixAutoSignal:= , 
	ixServiceSignal:= , 
	iiPLCMode:= PLC_Mode, 
	qxSignal=> );
	
// КОМАНДЫ - ЧРП
	
xVFD_Start(
	ixAutoSignal:= , 
	ixServiceSignal:= , 
	iiPLCMode:= PLC_Mode, 
	qxSignal=> );

xVFD_Stop(
	ixAutoSignal:= , 
	ixServiceSignal:= , 
	iiPLCMode:= PLC_Mode, 
	qxSignal=> );

xVFD_EmergencyStop(
	ixAutoSignal:= , 
	ixServiceSignal:= , 
	iiPLCMode:= PLC_Mode, 
	qxSignal=> );

xVFD_Reset(
	ixAutoSignal:= , 
	ixServiceSignal:= , 
	iiPLCMode:= PLC_Mode, 
	qxSignal=> );

// КОМАНДЫ - ЗРА

xBY_Open(
	ixAutoSignal:= , 
	ixServiceSignal:= , 
	iiPLCMode:= PLC_Mode, 
	qxSignal=> );
	
xBY_Close(
	ixAutoSignal:= , 
	ixServiceSignal:= , 
	iiPLCMode:= PLC_Mode, 
	qxSignal=> );

xBY_Stop(
	ixAutoSignal:= , 
	ixServiceSignal:= , 
	iiPLCMode:= PLC_Mode, 
	qxSignal=> );

xBY_Reset(
	ixAutoSignal:= , 
	ixServiceSignal:= , 
	iiPLCMode:= PLC_Mode, 
	qxSignal=> );

                        
END_METHOD

METHOD Process_VFD
VAR_INPUT
END_VAR
                          Process_VFD_qFreq();
Process_VFD_Commands(
	rtrig_vfdCmd_xStart.Q,
	rtrig_vfdCmd_xStop.Q,
	rtrig_vfdCmd_xEmergencyStop.Q,
	rtrig_vfdCmd_xReset.Q
);
Process_VFD_Signals();
                        
END_METHOD

METHOD Process_LifeBit
VAR_INPUT
END_VAR
                          
                        
END_METHOD

METHOD Process_BY_Commands
VAR_INPUT
	xOpen : BOOL;
	xClose : BOOL;
	xStop : BOOL;
	XReset : BOOL;
END_VAR
                          
                        
END_METHOD

METHOD Condition_BY_Open : BOOL
VAR_INPUT
	i : INT;
END_VAR
                          Condition_BY_Open := 
	NOT GetStatus_BY_Error(i)
	AND NOT GetStatus_BY_Open(i);
                        
END_METHOD

METHOD Condition_BY_Close : BOOL
VAR_INPUT
	i : INT;
END_VAR
                          Condition_BY_Open := 
	NOT GetStatus_BY_Error(i)
	AND NOT GetStatus_BY_Closed(i);
                        
END_METHOD

METHOD init_BY
VAR_INPUT
END_VAR
                          BY1(
	ixOpenCmd:= rtrig_byCmd_xOpen.Q AND by_iChange = 1, 
	ixCloseCmd:= rtrig_byCmd_xClose.Q AND by_iChange = 1, 
	ixStopCmd:= rtrig_byCmd_xStop.Q AND by_iChange = 1, 
	ixResetCmd:= rtrig_byCmd_xReset AND by_iChange =1, 
	ixReadyStatus:= GetStatus_BY_Ready(1), 
	ixErrorCommonStatus:= GetStatus_BY_Error(1), 
	ixManualStatus:= , 
	ixOpenStatus:= GetStatus_BY_Open(1), 
	ixClosedStatus:= GetStatus_BY_Closed(1), 
	qxOpen=> , 
	qxClose=> , 
	qxErrorCommonStatus=> , 
	qxManualStatus=> , 
	qxStoppedStatus=> , 
	qxOpenProcessStatus=> , 
	qxCloseProcessStatus=> , 
	qxOpenStatus=> , 
	qxClosedStatus=> );

BY2(
	ixOpenCmd := rtrig_byCmd_xOpen.Q AND by_iChange = 2,
	ixCloseCmd := rtrig_byCmd_xClose.Q AND by_iChange = 2,
	ixStopCmd := rtrig_byCmd_xStop.Q AND by_iChange = 2,
	ixResetCmd := rtrig_byCmd_xReset AND by_iChange = 2,
	ixReadyStatus := GetStatus_BY_Ready(2),
	ixErrorCommonStatus := GetStatus_BY_Error(2),
	ixManualStatus := ,
	ixOpenStatus := GetStatus_BY_Open(2),
	ixClosedStatus := GetStatus_BY_Closed(2),
	qxOpen => ,
	qxClose => ,
	qxErrorCommonStatus => ,
	qxManualStatus => ,
	qxStoppedStatus => ,
	qxOpenProcessStatus => ,
	qxCloseProcessStatus => ,
	qxOpenStatus => ,
	qxClosedStatus => );

BY3(
	ixOpenCmd := rtrig_byCmd_xOpen.Q AND by_iChange = 3,
	ixCloseCmd := rtrig_byCmd_xClose.Q AND by_iChange = 3,
	ixStopCmd := rtrig_byCmd_xStop.Q AND by_iChange = 3,
	ixResetCmd := rtrig_byCmd_xReset AND by_iChange = 3,
	ixReadyStatus := GetStatus_BY_Ready(3),
	ixErrorCommonStatus := GetStatus_BY_Error(3),
	ixManualStatus := ,
	ixOpenStatus := GetStatus_BY_Open(3),
	ixClosedStatus := GetStatus_BY_Closed(3),
	qxOpen => ,
	qxClose => ,
	qxErrorCommonStatus => ,
	qxManualStatus => ,
	qxStoppedStatus => ,
	qxOpenProcessStatus => ,
	qxCloseProcessStatus => ,
	qxOpenStatus => ,
	qxClosedStatus => );

BY4(
	ixOpenCmd := rtrig_byCmd_xOpen.Q AND by_iChange = 4,
	ixCloseCmd := rtrig_byCmd_xClose.Q AND by_iChange = 4,
	ixStopCmd := rtrig_byCmd_xStop.Q AND by_iChange = 4,
	ixResetCmd := rtrig_byCmd_xReset AND by_iChange = 4,
	ixReadyStatus := GetStatus_BY_Ready(4),
	ixErrorCommonStatus := GetStatus_BY_Error(4),
	ixManualStatus := ,
	ixOpenStatus := GetStatus_BY_Open(4),
	ixClosedStatus := GetStatus_BY_Closed(4),
	qxOpen => ,
	qxClose => ,
	qxErrorCommonStatus => ,
	qxManualStatus => ,
	qxStoppedStatus => ,
	qxOpenProcessStatus => ,
	qxCloseProcessStatus => ,
	qxOpenStatus => ,
	qxClosedStatus => );

BY5(
	ixOpenCmd := rtrig_byCmd_xOpen.Q AND by_iChange = 5,
	ixCloseCmd := rtrig_byCmd_xClose.Q AND by_iChange = 5,
	ixStopCmd := rtrig_byCmd_xStop.Q AND by_iChange = 5,
	ixResetCmd := rtrig_byCmd_xReset AND by_iChange = 5,
	ixReadyStatus := GetStatus_BY_Ready(5),
	ixErrorCommonStatus := GetStatus_BY_Error(5),
	ixManualStatus := ,
	ixOpenStatus := GetStatus_BY_Open(5),
	ixClosedStatus := GetStatus_BY_Closed(5),
	qxOpen => ,
	qxClose => ,
	qxErrorCommonStatus => ,
	qxManualStatus => ,
	qxStoppedStatus => ,
	qxOpenProcessStatus => ,
	qxCloseProcessStatus => ,
	qxOpenStatus => ,
	qxClosedStatus => );

BY7(
	ixOpenCmd := rtrig_byCmd_xOpen.Q AND by_iChange = 7,
	ixCloseCmd := rtrig_byCmd_xClose.Q AND by_iChange = 7,
	ixStopCmd := rtrig_byCmd_xStop.Q AND by_iChange = 7,
	ixResetCmd := rtrig_byCmd_xReset AND by_iChange = 7,
	ixReadyStatus := GetStatus_BY_Ready(7),
	ixErrorCommonStatus := GetStatus_BY_Error(7),
	ixManualStatus := ,
	ixOpenStatus := GetStatus_BY_Open(7),
	ixClosedStatus := GetStatus_BY_Closed(7),
	qxOpen => ,
	qxClose => ,
	qxErrorCommonStatus => ,
	qxManualStatus => ,
	qxStoppedStatus => ,
	qxOpenProcessStatus => ,
	qxCloseProcessStatus => ,
	qxOpenStatus => ,
	qxClosedStatus => );

BY8(
	ixOpenCmd := rtrig_byCmd_xOpen.Q AND by_iChange = 8,
	ixCloseCmd := rtrig_byCmd_xClose.Q AND by_iChange = 8,
	ixStopCmd := rtrig_byCmd_xStop.Q AND by_iChange = 8,
	ixResetCmd := rtrig_byCmd_xReset AND by_iChange = 8,
	ixReadyStatus := GetStatus_BY_Ready(8),
	ixErrorCommonStatus := GetStatus_BY_Error(8),
	ixManualStatus := ,
	ixOpenStatus := GetStatus_BY_Open(8),
	ixClosedStatus := GetStatus_BY_Closed(8),
	qxOpen => ,
	qxClose => ,
	qxErrorCommonStatus => ,
	qxManualStatus => ,
	qxStoppedStatus => ,
	qxOpenProcessStatus => ,
	qxCloseProcessStatus => ,
	qxOpenStatus => ,
	qxClosedStatus => );

                        
END_METHOD

METHOD Process_BY_Signals
VAR_INPUT
END_VAR
                          Set_BY_Open(1, BY1.qxOpen);
Set_BY_Close(1, BY1.qxClose);

Set_BY_Open(2, BY2.qxOpen);
Set_BY_Close(2, BY2.qxClose);

Set_BY_Open(3, BY3.qxOpen);
Set_BY_Close(3, BY3.qxClose);

Set_BY_Open(4, BY4.qxOpen);
Set_BY_Close(4, BY4.qxClose);

Set_BY_Open(5, BY5.qxOpen);
Set_BY_Close(5, BY5.qxClose);

Set_BY_Open(7, BY7.qxOpen);
Set_BY_Close(7, BY7.qxClose);

Set_BY_Open(8, BY8.qxOpen);
Set_BY_Close(8, BY8.qxClose);

                        
END_METHOD

METHOD GetValue_BY_Change : INT
VAR_INPUT
END_VAR
                          GetValue_BY_Change := by_iChange;
                        
END_METHOD

METHOD Set_BY_Stop
VAR_INPUT
	i : INT;
	x : BOOL;
END_VAR
                          IF x THEN
	Set_BY_Close(i, FALSE);
	Set_BY_Open(i, FALSE);
END_IF;
                        
END_METHOD
END_PROGRAM

FUNCTION_BLOCK FB_SignalSplit
VAR_INPUT
	ixAutoSignal : BOOL;
	ixServiceSignal : BOOL;
	iiPLCMode : INT;
END_VAR
VAR_OUTPUT
	qxSignal : BOOL;
END_VAR
VAR
END_VAR

                    CASE iiPLCMode OF
	0: qxSignal := ixAutoSignal;
	2: qxSignal := ixServiceSignal;
END_CASE;
                  
END_FUNCTION_BLOCK

FUNCTION_BLOCK FB_BitMask
VAR_INPUT
	X : ARRAY[0..15] OF BOOL;
END_VAR
VAR_OUTPUT
	W : WORD;
END_VAR
VAR
END_VAR

                    W.0 := X[0];
W.1 := X[1];
W.2 := X[2];
W.3 := X[3];
W.4 := X[4];
W.5 := X[5];
W.6 := X[6];
W.7 := X[7];
W.8 := X[8];
W.9 := X[9];
W.10 := X[10];
W.11 := X[11];
W.12 := X[12];
W.13 := X[13];
W.14 := X[14];
W.15 := X[15];

                  
END_FUNCTION_BLOCK

FUNCTION_BLOCK FB_Shutter IMPLEMENTS IShutterCommands, IShutterFeedback
VAR_INPUT
	ixOpenCmd : BOOL;	// Команда открыть
	ixCloseCmd : BOOL;	// Команда закрыть
	ixStopCmd : BOOL;	// Команда остановить
	ixResetCmd : BOOL;	// Сброс всех ошибок
	
	ixReadyStatus : BOOL;	// Состояние - готов.
	ixErrorCommonStatus : BOOL;	// Авария - обобщённая
	ixManualStatus : BOOL;	// ЗРА в местном управлении
	ixOpenStatus : BOOL;	// Статус - открыт
	ixClosedStatus : BOOL; 	// Статус - закрыт
END_VAR
VAR_OUTPUT
	qxOpen : BOOL;		// Открытие затвора
	qxClose : BOOL;		// Закрытие затвора
	
	qxErrorCommonStatus : BOOL; 	// Транзит сигнала ошибки ЗРА
	qxManualStatus : BOOL;			// Транзит сигнала ручного управления
	qxStoppedStatus : BOOL;			// Сигнал ЗРА остановлен
	qxOpenProcessStatus : BOOL;		// Процесс открытия затвора
	qxCloseProcessStatus : BOOL;	// Процесс закрытия затвора
	qxOpenStatus : BOOL;	// Статус - открыт
	qxClosedStatus : BOOL; 	// Статус - закрыт
END_VAR
VAR
END_VAR

                    UpdateFeedbackProcess();
CloseOpenProcess();
                  

METHOD UpdateFeedbackProcess : BOOL
VAR_INPUT
END_VAR
VAR
	ftrig_qxOpenProcessStatus : F_TRIG;
	ftrig_qxCloseProcessStatus : F_TRIG;
END_VAR
                          ftrig_qxOpenProcessStatus(CLK:= qxOpen, Q=> );
ftrig_qxCloseProcessStatus(CLK:= qxClose, Q=> );

IF ftrig_qxOpenProcessStatus.Q THEN qxOpenProcessStatus := FALSE; END_IF;
IF ftrig_qxCloseProcessStatus.Q THEN qxCloseProcessStatus := FALSE; END_IF;

qxOpenStatus := GetStatusOpen();
qxClosedStatus := GetStatusClosed();

qxManualStatus := GetStatusManual();

qxErrorCommonStatus := GetStatusCommonError();

                        
END_METHOD

METHOD CloseOpenProcess : BOOL
VAR_INPUT
END_VAR
VAR
	xOpen : BOOL;
	xClose : BOOL;
	
	rtrig_ixOpenCmd : R_TRIG;
	rtrig_ixCloseCmd : R_TRIG;
	rtrig_ixStopCmd : R_TRIG;
	rtrig_ixResetCmd : R_TRIG;
	
	rtrig_ixOpenStatus : R_TRIG;
	rtrig_ixClosedStatus : R_TRIG;
	
END_VAR
                          rtrig_ixOpenCmd(CLK:= ixOpenCmd, Q=> );
rtrig_ixCloseCmd(CLK:= ixCloseCmd, Q=> );
rtrig_ixStopCmd(CLK:= ixStopCmd, Q=> );
rtrig_ixResetCmd(CLK:= ixResetCmd, Q=> );

rtrig_ixOpenStatus(CLK:= ixOpenStatus, Q=> );
rtrig_ixClosedStatus(CLK:= ixClosedStatus, Q=> );

IF NOT GetStatusManual() THEN
	IF rtrig_ixOpenCmd.Q AND GetStatusReady() AND NOT GetStatusOpen() THEN
		cmdOpen(TRUE);
	END_IF;
	
	IF rtrig_ixCloseCmd.Q AND GetStatusReady() AND NOT GetStatusClosed() THEN
		cmdClose(TRUE);
	END_IF;
	
	IF OpenCloseProcessStatus() AND GetStatusOpen() THEN
		cmdOpen(FALSE);
	END_IF;
	
	IF OpenCloseProcessStatus() AND GetStatusClosed() THEN
		cmdClose(FALSE);
	END_IF;
	
	IF rtrig_ixStopCmd.Q THEN
		cmdStop(TRUE);
	END_IF;
	
	IF rtrig_ixResetCmd.Q THEN cmdReset(); END_IF;

END_IF;
                        
END_METHOD

METHOD OpenCloseProcessStatus : BOOL
VAR_INPUT
END_VAR
                          OpenCloseProcessStatus := qxOpen OR qxClose;
                        
END_METHOD

{warning 'добавить реализацию метода'}
METHOD GetStatusClosed : BOOL
VAR_INPUT
END_VAR
                          GetStatusClosed := ixClosedStatus;
                        
END_METHOD

{warning 'добавить реализацию метода'}
METHOD GetStatusCommonError : BOOL
VAR_INPUT
END_VAR
                          GetStatusCommonError := ixErrorCommonStatus;
                        
END_METHOD

{warning 'добавить реализацию метода'}
METHOD GetStatusManual : BOOL
VAR_INPUT
END_VAR
                          GetStatusManual := ixManualStatus;
                        
END_METHOD

{warning 'добавить реализацию метода'}
METHOD GetStatusOpen : BOOL
VAR_INPUT
END_VAR
                          GetStatusOpen := ixOpenStatus;
                        
END_METHOD

{warning 'добавить реализацию метода'}
METHOD GetStatusReady : BOOL
VAR_INPUT
END_VAR
                          GetStatusReady := ixReadyStatus;
                        
END_METHOD

{warning 'добавить реализацию метода'}
METHOD cmdClose : BOOL
VAR_INPUT
	xClose : BOOL;
END_VAR
VAR
END_VAR
                          IF xClose THEN
	qxClose := TRUE;
	qxCloseProcessStatus := TRUE;
	qxStoppedStatus := FALSE;
ELSIF NOT xClose THEN
	qxClose := FALSE;
	qxCloseProcessStatus := FALSE;
END_IF;
                        
END_METHOD

{warning 'добавить реализацию метода'}
METHOD cmdOpen : BOOL
VAR_INPUT
	xOpen	: BOOL;
END_VAR
                          IF xOpen THEN
	qxOpen := TRUE;
	qxOpenProcessStatus := TRUE;
	qxStoppedStatus := FALSE;
ELSIF NOT xOpen THEN
	qxOpen := FALSE;
	qxOpenProcessStatus := FALSE;
END_IF;
                        
END_METHOD

{warning 'добавить реализацию метода'}
METHOD cmdReset : BOOL
VAR_INPUT
END_VAR
                          qxErrorCommonStatus := FALSE;
                        
END_METHOD

{warning 'добавить реализацию метода'}
METHOD cmdStop : BOOL
VAR_INPUT
	xStop	: BOOL;
END_VAR
                          IF xStop THEN
	cmdClose(FALSE);
	cmdOpen(FALSE);
	qxStoppedStatus := TRUE;
END_IF;
                        
END_METHOD
END_FUNCTION_BLOCK

CONFIGURATION Device
  RESOURCE Application ON PLC
(* global variable list TargetVars *)
{attribute 'qualified_only'}
VAR_GLOBAL
	stBuzzer:	 TRG_Buzzer;
	stDebug: 	 TRG_Debug;
	stDrives: 	 TRG_Drives;
	stRtc:		 TRG_RTC;
	stInfo:		 TRG_Info;
	stWatchdog:	 TRG_Watchdog;
	stPlc210:	 TRG_PLC210;
	stLeftSide:	 TRG_LeftSide;
	stRightSide: TRG_RightSide;
END_VAR
    TASK MainTask(INTERVAL := T#10ms, PRIORITY := 1);
    TASK VISU_TASK(INTERVAL := T#100ms, PRIORITY := 31);
    TASK SoftMotion_PlanningTask(INTERVAL := T#2ms, PRIORITY := 15);
    PROGRAM LEGACY_MAIN WITH MainTask : LEGACY_MAIN;
    PROGRAM VisuElems.Visu_Prg WITH VISU_TASK : VisuElems.Visu_Prg;
  END_RESOURCE
END_CONFIGURATION

CONFIGURATION Ethernet_1
END_CONFIGURATION

CONFIGURATION ModbusTCP_Slave_Device_1
END_CONFIGURATION

CONFIGURATION Modbus_TCP_Master_1
END_CONFIGURATION

CONFIGURATION MV210_202_1A3
END_CONFIGURATION

CONFIGURATION MV210_202_1A4
END_CONFIGURATION

CONFIGURATION MV210_202_1A5
END_CONFIGURATION

CONFIGURATION MU210_403_1A6
END_CONFIGURATION

CONFIGURATION MV210_101_1A7
END_CONFIGURATION

CONFIGURATION MU210_502_1A8
END_CONFIGURATION

CONFIGURATION MV210_202_1A2
END_CONFIGURATION

CONFIGURATION Modbus_COM
END_CONFIGURATION

CONFIGURATION Modbus_Master_COM_Port
END_CONFIGURATION

CONFIGURATION TKC1
END_CONFIGURATION

CONFIGURATION TKC2
END_CONFIGURATION

CONFIGURATION _1UZ8
END_CONFIGURATION

CONFIGURATION _2UZ8
END_CONFIGURATION

CONFIGURATION Modbus_COM_1
END_CONFIGURATION

CONFIGURATION Modbus_Master_COM_Port_1
END_CONFIGURATION

CONFIGURATION _0303_05_BY01_modbusSlave
END_CONFIGURATION

CONFIGURATION _0303_05_BY02_modbusSlave
END_CONFIGURATION

CONFIGURATION _0303_05_BY03_modbusSlave
END_CONFIGURATION

CONFIGURATION _0303_05_BY04_modbusSlave
END_CONFIGURATION

CONFIGURATION _0303_05_BY05_modbusSlave
END_CONFIGURATION

CONFIGURATION _0303_05_BY07_modbusSlave
END_CONFIGURATION

CONFIGURATION _0303_05_BY08_modbusSlave
END_CONFIGURATION
